// TIA Portal V19 export
DATA_BLOCK "RO PROCESS"   // DB105
{ S7_Optimized_Access := 'TRUE' }
// stored: MemoryReserve 100
   VAR
      RO : Int;
      "ORP SET VALUE" : Int;
      "PRESSURE SET POINT" : Int;
      "ORP BUFF" : Int;
      OUTPUT : Struct
         "ORP AV-1" : Bool;
         "RO FEED PUMP" : Bool;
         "DP-2" : Bool;
         "DP-5" : Bool;
         "DP-6" : Bool;
         "RO-1 HPP PUMP" : Bool;
         UV : Bool;
         "RO-2 HPP PUMP" : Bool;
      END_STRUCT;
   END_VAR
BEGIN
END_DATA_BLOCK
